// Mitsubishi GX Developer project: 10-805培林與軸套自動壓合機   PLC: FX1N

PROGRAM MAIN
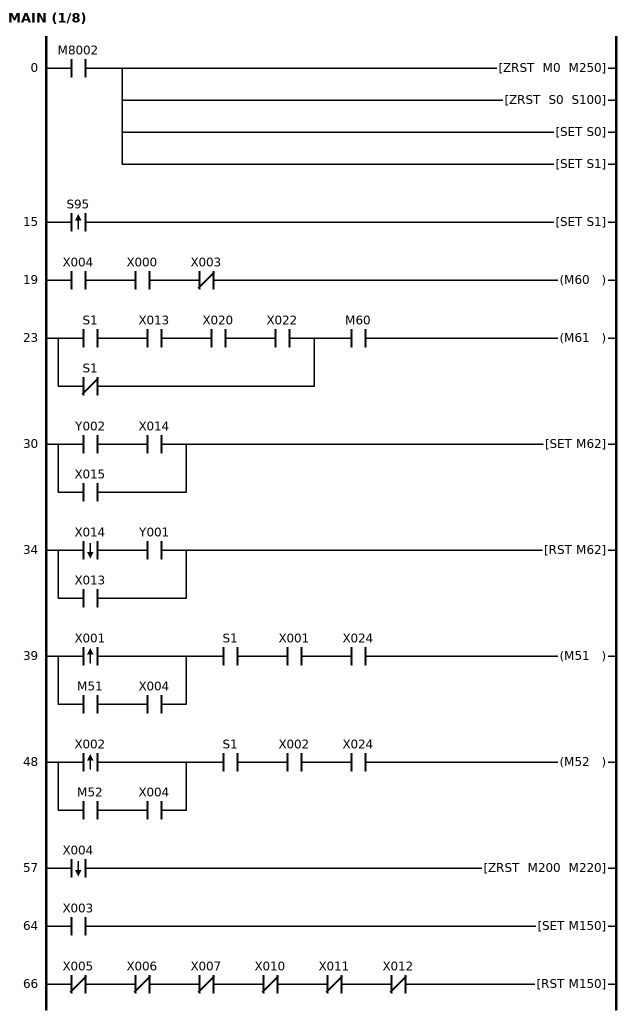
0     LD      M8002
      ZRST    M0 M250
      ZRST    S0 S100
      SET     S0
      SET     S1
15    LDP     S95
      SET     S1
19    LD      X004
      AND     X000
      ANI     X003
      OUT     M60
23    LD      S1
      AND     X013
      AND     X020
      AND     X022
      ORI     S1
      AND     M60
      OUT     M61
30    LD      Y002
      AND     X014
      OR      X015
      SET     M62
34    LDF     X014
      AND     Y001
      OR      X013
      RST     M62
39    LDP     X001
      LD      M51
      AND     X004
      ORB
      AND     S1
      AND     X001
      AND     X024
      OUT     M51
48    LDP     X002
      LD      M52
      AND     X004
      ORB
      AND     S1
      AND     X002
      AND     X024
      OUT     M52
57    LDF     X004
      ZRST    M200 M220
64    LD      X003
      SET     M150
66    LDI     X005
      ANI     X006
      ANI     X007
      ANI     X010
      ANI     X011
      ANI     X012
      RST     M150
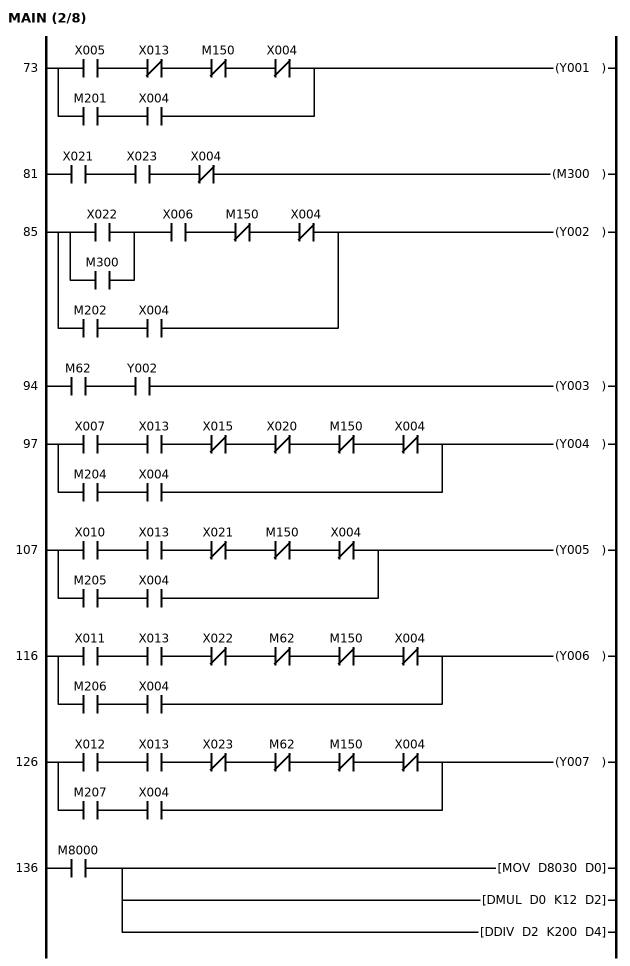
73    LD      X005
      ANI     X013
      ANI     M150
      ANI     X004
      LD      M201
      AND     X004
      ORB
      OUT     Y001
81    LD      X021
      AND     X023
      ANI     X004
      OUT     M300
85    LD      X022
      OR      M300
      AND     X006
      ANI     M150
      ANI     X004
      LD      M202
      AND     X004
      ORB
      OUT     Y002
94    LD      M62
      AND     Y002
      OUT     Y003
97    LD      X007
      AND     X013
      ANI     X015
      ANI     X020
      ANI     M150
      ANI     X004
      LD      M204
      AND     X004
      ORB
      OUT     Y004
107   LD      X010
      AND     X013
      ANI     X021
      ANI     M150
      ANI     X004
      LD      M205
      AND     X004
      ORB
      OUT     Y005
116   LD      X011
      AND     X013
      ANI     X022
      ANI     M62
      ANI     M150
      ANI     X004
      LD      M206
      AND     X004
      ORB
      OUT     Y006
126   LD      X012
      AND     X013
      ANI     X023
      ANI     M62
      ANI     M150
      ANI     X004
      LD      M207
      AND     X004
      ORB
      OUT     Y007
136   LD      M8000
      MOV     D8030 D0
      DMUL    D0 K12 D2
      DDIV    D2 K200 D4
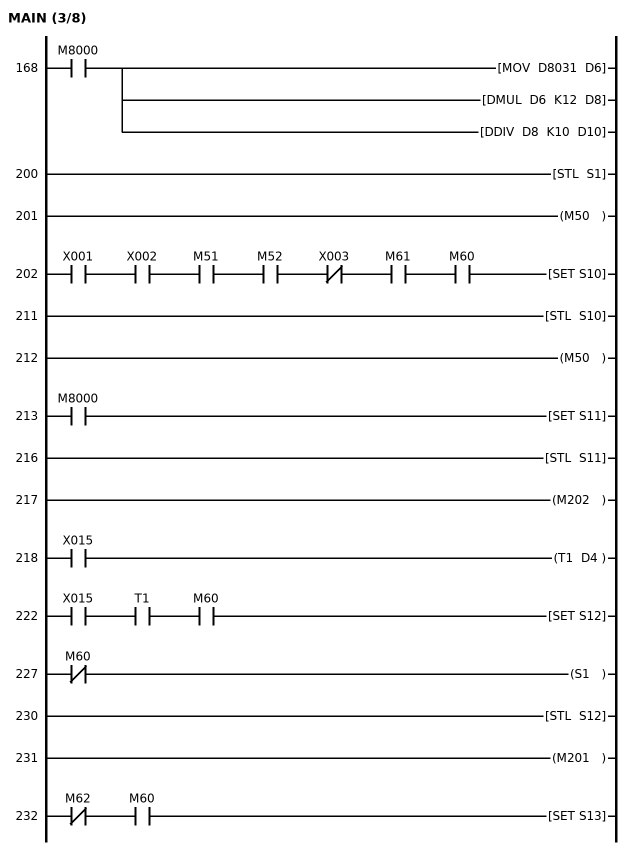
168   LD      M8000
      MOV     D8031 D6
      DMUL    D6 K12 D8
      DDIV    D8 K10 D10
200   STL     S1
201   OUT     M50
202   LD      X001
      AND     X002
      AND     M51
      AND     M52
      ANI     X003
      AND     M61
      AND     M60
      SET     S10
211   STL     S10
212   OUT     M50
213   LD      M8000
      SET     S11
216   STL     S11
217   OUT     M202
218   LD      X015
      OUT     T1 D4
222   LD      X015
      AND     T1
      AND     M60
      SET     S12
227   LDI     M60
      OUT     S1
230   STL     S12
231   OUT     M201
232   LDI     M62
      AND     M60
      SET     S13
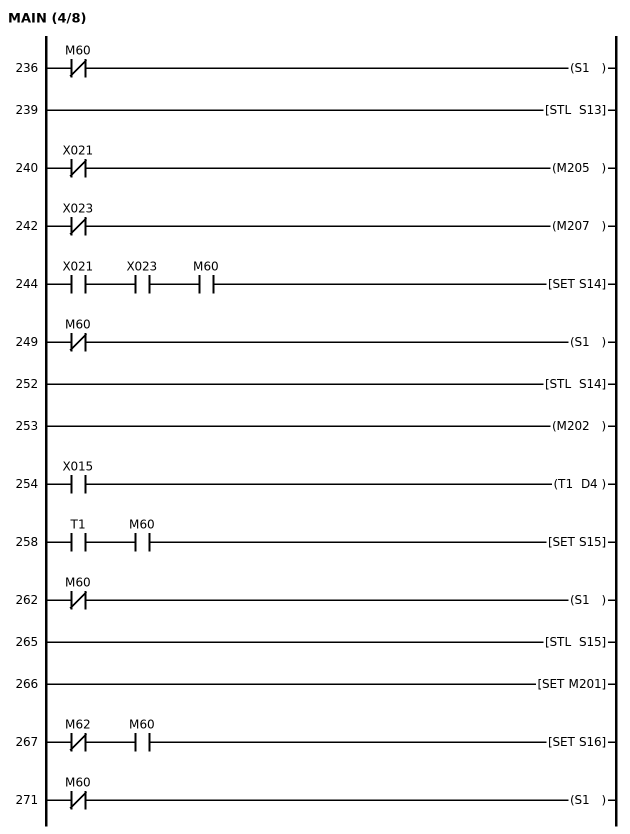
236   LDI     M60
      OUT     S1
239   STL     S13
240   LDI     X021
      OUT     M205
242   LDI     X023
      OUT     M207
244   LD      X021
      AND     X023
      AND     M60
      SET     S14
249   LDI     M60
      OUT     S1
252   STL     S14
253   OUT     M202
254   LD      X015
      OUT     T1 D4
258   LD      T1
      AND     M60
      SET     S15
262   LDI     M60
      OUT     S1
265   STL     S15
266   SET     M201
267   LDI     M62
      AND     M60
      SET     S16
271   LDI     M60
      OUT     S1
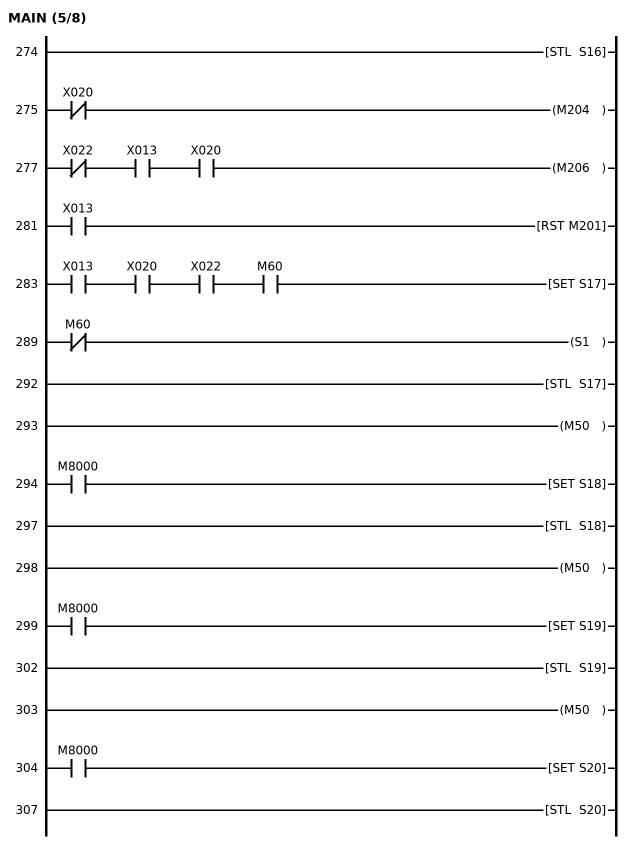
274   STL     S16
275   LDI     X020
      OUT     M204
277   LDI     X022
      AND     X013
      AND     X020
      OUT     M206
281   LD      X013
      RST     M201
283   LD      X013
      AND     X020
      AND     X022
      AND     M60
      SET     S17
289   LDI     M60
      OUT     S1
292   STL     S17
293   OUT     M50
294   LD      M8000
      SET     S18
297   STL     S18
298   OUT     M50
299   LD      M8000
      SET     S19
302   STL     S19
303   OUT     M50
304   LD      M8000
      SET     S20
307   STL     S20
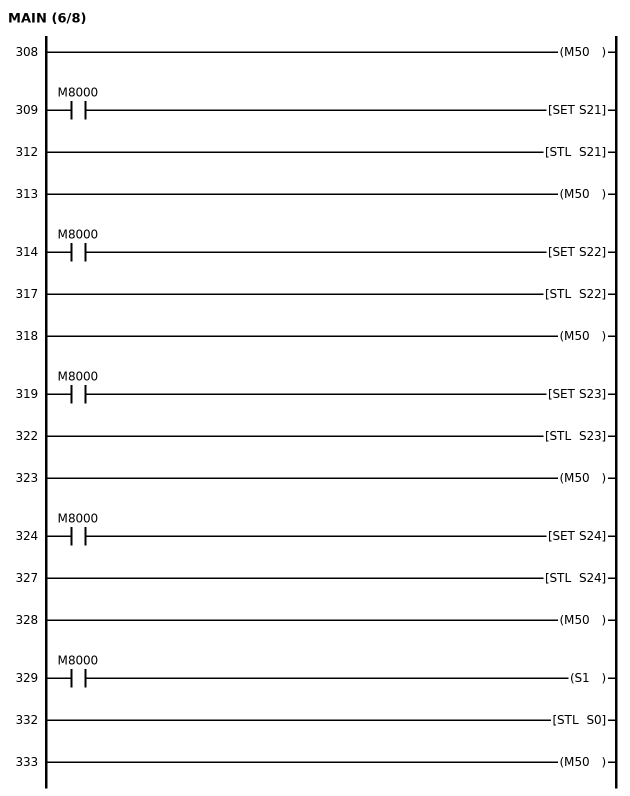
308   OUT     M50
309   LD      M8000
      SET     S21
312   STL     S21
313   OUT     M50
314   LD      M8000
      SET     S22
317   STL     S22
318   OUT     M50
319   LD      M8000
      SET     S23
322   STL     S23
323   OUT     M50
324   LD      M8000
      SET     S24
327   STL     S24
328   OUT     M50
329   LD      M8000
      OUT     S1
332   STL     S0
333   OUT     M50
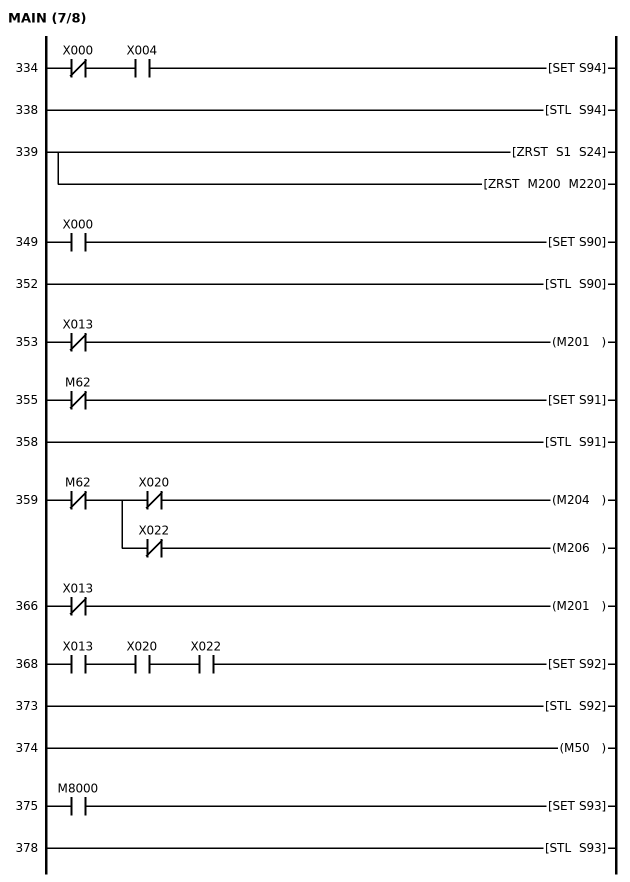
334   LDI     X000
      AND     X004
      SET     S94
338   STL     S94
339   ZRST    S1 S24
      ZRST    M200 M220
349   LD      X000
      SET     S90
352   STL     S90
353   LDI     X013
      OUT     M201
355   LDI     M62
      SET     S91
358   STL     S91
359   LDI     M62
      MPS
      ANI     X020
      OUT     M204
      MPP
      ANI     X022
      OUT     M206
366   LDI     X013
      OUT     M201
368   LD      X013
      AND     X020
      AND     X022
      SET     S92
373   STL     S92
374   OUT     M50
375   LD      M8000
      SET     S93
378   STL     S93
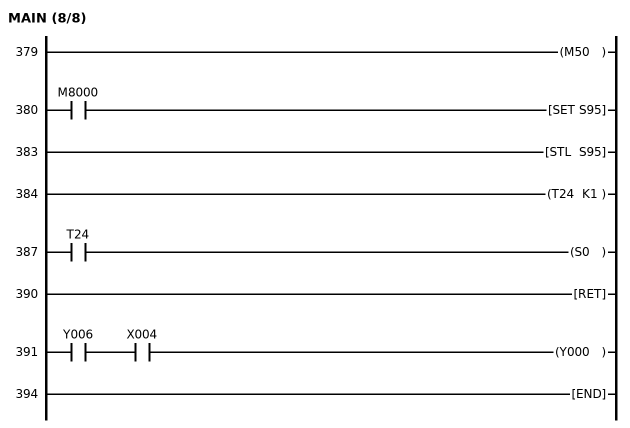
379   OUT     M50
380   LD      M8000
      SET     S95
383   STL     S95
384   OUT     T24 K1
387   LD      T24
      OUT     S0
390   RET
391   LD      Y006
      AND     X004
      OUT     Y000
394   END
END_PROGRAM
